VAR_OUTPUT
	Error: BOOL;
	errorID: UDINT;
END_VAR
MCPOS(Axis:=Axis,Error=>Error,ErrorID=>errorID);
END_METHOD

METHOD setReset : BOOL
VAR_INPUT
END_VAR
END_METHOD

METHOD setStop : BOOL
VAR_INPUT
END_VAR
velocityEnable:=FALSE;
stopEnable:=TRUE;
haltEnable:=FALSE;
homeEnable:= FALSE;
torqueEnable:= FALSE;
posEnable:=FALSE;
END_METHOD

METHOD setTorque : BOOL
VAR_INPUT
END_VAR
velocityEnable:=FALSE;
stopEnable:=FALSE;
haltEnable:=FALSE;
homeEnable:= FALSE;
torqueEnable:= TRUE;
posEnable:=FALSE;
END_METHOD

METHOD setVelocity : BOOL
VAR_INPUT
END_VAR
velocityEnable:=TRUE;
stopEnable:=FALSE;
haltEnable:=FALSE;
homeEnable:= FALSE;
torqueEnable:= FALSE;
posEnable:=FALSE;
END_METHOD

METHOD stateUpdate : BOOL
VAR_INPUT
END_VAR
IF powerEnable OR haltEnable OR stopEnable THEN
	state:=1;
END_IF
IF NOT enabled THEN
	state:=2;
END_IF
IF torqueEnable OR velocityEnable OR posEnable THEN
	state:=3;
END_IF
IF AXIS.Status.Error THEN
	state:=4;
END_IF
END_METHOD

METHOD stop_error_check : BOOL
VAR_INPUT
END_VAR

VAR_OUTPUT
	errorID: UDINT;
	Error: BOOL;
END_VAR
MCSTOP(Axis:=Axis,Error=>Error,ErrorID=>errorID);
END_METHOD

METHOD torque_error_check : BOOL
VAR_INPUT
END_VAR

VAR_OUTPUT
	Error: BOOL;
	errorID: UDINT;
END_VAR
MCTORQUECONTROL(Axis:=Axis,Error=>Error,ErrorID=>errorID);
END_METHOD

METHOD velocity_error_check : BOOL
VAR_INPUT
END_VAR

VAR_OUTPUT
	Error: BOOL;
	errorID: UDINT;
END_VAR
MCVELOCITY(Axis:=Axis,Error=>Error,ErrorID=>errorID);
END_METHOD

END_FUNCTION_BLOCK
